# EPICS substitutions: axisApp/Db/axis.substitutions
# Set points do not have units set because it will cause it to be processed thus sending a possibly wrong value
# to the display

file $(UTILITIES)/db/unit_setter.template {
  pattern
    {P,    FROM, TO, PROCESS_FLAGS}

    {"\$(P)", "\$(mAXIS).EGU", "\$(AXIS)", "PP"}
    {"\$(P)", "\$(mAXIS).EGU", "\$(AXIS):SP:RBV", "PP"}
    {"\$(P)", "\$(mAXIS).EGU", "\$(AXIS):SP", "NPP"}
}

file axis_base.template {
  pattern
    {P,    mAXIS, AXIS}

    {"\$(P)", "\$(mAXIS)", "\$(AXIS)"}
}
